(* IEC 61131-3 sources: POMIRTS_lab3/AS/Library/AsBrWStr, 2 files *)

(* ---- AsBrWStr.fun ---- *)
(********************************************************************
 * COPYRIGHT -- Bernecker + Rainer
 ********************************************************************
 * Library: AsBrWStr
 * File: AsBrWStr.fun
 * Author: B+R
 ********************************************************************
 * Functions and function blocks of library AsBrWStr
 ********************************************************************)

FUNCTION brwcsconv : UDINT						(*converts one string to a different format*)
	VAR_INPUT
		pDestination	:REFERENCE TO USINT;	(*string to be appended to, given as a pointer*)
		pSource	:REFERENCE TO USINT;			(*string to be appended, given as a pointer*)
		level	:USINT;							(*brwU8toUC (= 0) if converting from U8 to UC; brwUCtoU8 (= 1) if converting from UC to U8*)
	END_VAR
END_FUNCTION
FUNCTION brwcsncpy : UDINT						(*copies a maximum of n characters from the pSource WC string to the pDestination address*)
	VAR_INPUT
		pDestination	:REFERENCE TO UINT;		(*pointer to the target memory for the string*)
		pSource	:REFERENCE TO UINT;				(*string to be copied, given as a pointer*)
		n	:UDINT;								(*max. number of characters to be copied*)
	END_VAR
END_FUNCTION
FUNCTION brwcsncat : UDINT						(*appends a maximum of n characters from the pSource string to the pDestination string*)
	VAR_INPUT
		pDestination	:REFERENCE TO UINT;		(*string to be appended to, given as a pointer*)
		pSource	:REFERENCE TO UINT;				(*string to be appended, given as a pointer*)
		n	:UDINT;								(*maximum number of characters to be added from pSource to pDestination*)
	END_VAR
END_FUNCTION
FUNCTION brwcscat : UDINT						(*connects two WC strings to each other (concatenation)*)
	VAR_INPUT
		pDestination	:REFERENCE TO UINT;		(*string to be appended to, given as a pointer*)
		pSource	:REFERENCE TO UINT;				(*string to be appended, given as a pointer*)
	END_VAR
END_FUNCTION
FUNCTION brwcscmp : DINT						(*compares two 16-bit character strings*)
	VAR_INPUT
		pUcstr1	:REFERENCE TO UINT;				(*first string, given as a pointer*)
		pUcstr2	:REFERENCE TO UINT;				(*second string, given as a pointer*)
	END_VAR
END_FUNCTION
FUNCTION brwcslen : UDINT						(*determines the length of a WC string*)
	VAR_INPUT
		pwcString	:REFERENCE TO UINT;			(*string whose length should be determined, given as a pointer*)
	END_VAR
END_FUNCTION
FUNCTION brwcsset : UDINT						(*appends the pSource string to the pDestination string*)
	VAR_INPUT
		pDestination	:REFERENCE TO UINT;		(*string being written, given as a pointer*)
		len	:UDINT;								(*number of characters to be written*)
		symbol	:UINT;							(*character used to overwrite*)
	END_VAR
END_FUNCTION
FUNCTION brwcsncmp : DINT						(*compares two 16-bit strings*)
	VAR_INPUT
		pwcString1	:REFERENCE TO UINT;			(*first string given as a pointer*)
		pwcString2	:REFERENCE TO UINT;			(*second string given as a pointer*)
		n	:UDINT;								(*max. number of characters from pUcstr1 to be compared with pUcstr2*)
	END_VAR
END_FUNCTION
FUNCTION brwcscpy : UDINT						(*copies a WC string*)
	VAR_INPUT
		pDestination	:REFERENCE TO UINT;		(*pointer to the target memory for the string*)
		pSource	:REFERENCE TO UINT;				(*string to be copied, given as a pointer*)
	END_VAR
END_FUNCTION
FUNCTION brwcsrchr : UDINT						(*searches for the last occurrence of a certain character in a WC string*)
	VAR_INPUT
		pDestination	:REFERENCE TO UINT;		(*character string being searched, given as a pointer*)
		symbol	:UINT;							(*character being looked for*)
	END_VAR
END_FUNCTION
FUNCTION brwcschr : UDINT						(*searches for the first occurrence of a certain character*)
	VAR_INPUT
		pDestination	:REFERENCE TO UINT;		(*string given as a pointer*)
		symbol	:UINT;							(*character being looked for*)
	END_VAR
END_FUNCTION

(* ---- AsBrWStr.var ---- *)
(********************************************************************
 * COPYRIGHT -- Bernecker + Rainer
 ********************************************************************
 * Library: AsBrWStr
 * File: AsBrWStr.var
 * Author: B+R
 ********************************************************************
 * Local variables of library AsBrWStr
 ********************************************************************)

VAR CONSTANT
	brwUCtoU8	: USINT	:= 1;		(*instructs the wcsconv function to convert an ANSI character string into a WC string*)
	brwU8toUC	: USINT	:= 0;		(*instructs the wcsconv function to convert a WC character string into an ANSI string*)
END_VAR
